{attribute 'qualified_only'}
{attribute 'strict'}
{attribute 'to_string'}
TYPE E_Error :
(
	None		:= 0,
    Pause       := 4,	
    Hold      	:= 8,
	Complete	:= 16,	
	Stop		:= 32,
	Abort       := 64
);
END_TYPE

(* stored: Version 1.1.0.1
   DUT E_Error: Id {f95eda16-37d9-008f-37a3-b33cbc3ae97e} *)
